# B&R Automation Studio project ARuser
Automation Studio 4.10.4.38 SP; technology packages: mapp 5.17.0, mappView 5.17.0

## Configuration PC

CPU PC_any, AutomationRuntime D4.91, Build 4.1.2, Safety 0.0, Vc V4.52.0

### Task classes (Cpu.sw)
```
Cyclic#1 (cycle 10000 us):
  UserManage <- UserManagement.prg
Binaries: mvLoader, TCData, udbdef, User, asfw, OpcUaMap, iomap, sysconf, arconfig, ashwd, Role, ashwac
Libraries: ArUser, runtime, asieccon, astime, fileio, AsBrStr
```

### Hardware
```
PC : PC_any v1.1.1.0 (OrderNumber=PC)
  Connector IF3:
    InaPort = 11159
  ConfigurationID = ARuser_PC
  VolatileGlobalPvSize = 200000
  Cyclic1Duration = 10000
  Cyclic3Tolerance = 60000000
  Cyclic8Duration = 10000
  FileDevice1
  FileDeviceName1 = FileDevice
  FileDevicePath1 = C:\Users\hendricksf\Desktop
  ActivateOpcUa = 1
  OpcUaInformationModels_PV_Version = 1
```

### Config.mpuserx - PC/mappServices/Config.mpuserx
```
Element UserMgmtX (Type=mpuserx)
  Mgr:
    EditSameLevel = TRUE
  ServerSettings:
    Server:
      AdditionalUserData:
        [0] = mail
        [1] = telephoneNumber
  Users:
    DefUser#1:
      id = Anonymous
      name = 
    DefUser#2:
      id = Bob
      name = Bob Ross
    DefUser#3:
      id = Dave
      name = Dave Chapelle
    DefUser#4:
      id = John
      name = John Doe
  Groups:
    DefGroup#1:
      id = Everyone
      level = 1
    DefGroup#2:
      id = Operator
      level = 2
    DefGroup#3:
      id = Service
      level = 5
    DefGroup#4:
      id = Administrators
      admin = TRUE
```

## Configuration X20CP

CPU X20CP3585, AutomationRuntime D4.91, Build 4.1.2, Vc V4.52.0

### Task classes (Cpu.sw)
```
Cyclic#8:
  UserManage <- mappUser.UserManagement.prg
  RFIDdevice <- mappUser.RFIDdevice.prg
Libraries: runtime, standard, dvframe, sys_lib, AsUSB
```

### Task classes (Cpu.sw)
```
Cyclic#8:
  UserManage <- mappUser.UserManagement.prg
  RFIDdevice <- mappUser.RFIDdevice.prg
Binaries: mvLoader, udbdef, TCData, arconfig, User, Role, Config, iomap, asfw, ashwac, ashwd, sysconf
Libraries: runtime, standard, dvframe, sys_lib, AsUSB, operator, astime, AsIecCon, ArUser, AsBrStr, IecCheck, arssl, fileio, MpUserX, MpBase
```

### Hardware
```
X20CP3585 : X20CP3585 v1.5.0.0
  Connector IF2:
    ActivateDevice = 1
  ConfigurationID = ARuser_X20CP
  UserPartitionSize = 16
  VolatileGlobalPvSize = 120000
  ActivateOpcUa = 1
  OpcUaInformationModels_PV_Version = 1
```

## Logical view

Binary libraries used (declarations not repeated): operator, runtime, astime, AsIecCon, ArUser, AsBrStr, dvframe, AsUSB, sys_lib, standard, IecCheck, MpUserX 5.17.0, MpBase 5.17.0

### Global.typ - Globale Datentypen
```iecst
TYPE
	UserManagementEnum :
		(
		IdleState,
		DestroyListState,
		CreateUserState,
		DeleteUserState,
		ExportListState,
		ImportListState,
		ChangePasswordState,
		ComparePasswordState,
		CreateUserListGetNextState,
		CreateUserListGetFirstState,
		AssignRoleState,
		RoleListMainState,
		RoleListDeleteListState,
		RoleListInitListState,
		ErrorState,
		CreateRoleListGetFirstState,
		CreateRoleListGetNextState,
		RoleListGetNextState
		);
	typUSER : 	STRUCT
		CMD : typUSER_CMD;
		PAR : typUSER_PAR;
		DAT : typUSER_DAT;
		VIS : typUSER_VIS;
		ERR : typUSER_ERR;
	END_STRUCT;
	typUSER_CMD : 	STRUCT
		UserCreate : BOOL;
		UserDelete : BOOL;
		PasswordChange : BOOL;
		RoleCreate : BOOL;
		RoleDelete : BOOL;
		RoleAssign : BOOL;
		Import : BOOL;
		Export : BOOL;
		ListRefresh : BOOL;
		ErrorReset : BOOL;
	END_STRUCT;
	typUSER_PAR : 	STRUCT
		FilePath : STRING[80];
		UserName : STRING[40];
		UserRole : STRING[40];
		Password : STRING[40];
		PasswordRepeat : STRING[40];
		NumberOfUsers : USINT;
	END_STRUCT;
	typUSER_DAT : 	STRUCT
		Users : ARRAY[0..MaxUserNames]OF typUSER_DETAILS;
		Roles : ARRAY[0..MaxUserRoles]OF STRING[40];
		Status : STRING[80];
	END_STRUCT;
	typUSER_VIS : 	STRUCT
		ListUsers : ARRAY[0..MaxUserNames]OF STRING[80];
		ListUserIndex : UINT;
		ListUserRole : ARRAY[0..MaxUserRoles]OF STRING[80];
		ListUserRoleIndex : UINT;
		ListRoles : ARRAY[0..MaxUserRoles]OF STRING[80];
		ListRoleIndex : UINT;
	END_STRUCT;
	typUSER_ERR : 	STRUCT
		Number : DINT;
		State : UserManagementEnum;
	END_STRUCT;
	typUSER_DETAILS : 	STRUCT
		Roles : ARRAY[0..9]OF STRING[40];
		Name : STRING[40];
	END_STRUCT;
END_TYPE
```

### Global.var - Globale Variablen
```iecst
VAR
	ArUser : typUSER; (*Type for user data management*)
END_VAR
VAR CONSTANT
	MaxUserRoles : USINT := 20;
	MaxUserNames : USINT := 50;
END_VAR
```

### Package Logical/Libraries - Globale Bibliotheken

- Visualisation Logical/mappView (not shown)

### UserTypes.typ
```iecst
TYPE
	ClientInfoType : 	STRUCT
		userId : WSTRING[80];
		isValid : BOOL;
		ipAddress : WSTRING[15];
		languageId : WSTRING[2];
		screenResolution : WSTRING[32];
		slotId : SINT;
	END_STRUCT;
	rfidManagementEnum :
		(
		IdleRFID, (*Search for reader or new tokens*)
		SetToken, (*Assign token to user*)
		SetPassword, (*Set token as user password*)
		DeleteToken, (*Delete token from user*)
		IdentifyToken, (*Identify token*)
		CreateNodeList, (* Create a list of Node-IDs from all active USB devices*)
		ReadDeviceData, (* Read out the specific data from the Node-IDs*)
		CheckDevice, (* Check RFID reader data*)
		OpenDevice, (*Open serial communication*)
		InitDevice, (*Send inital data to setup RFID reader*)
		DataWrite, (*Send data to RFID reader*)
		DataRead, (*Read data from RFID reader*)
		CloseDevice, (*Close serial connection*)
		ErrorRFID (*Error state*)
		);
	enumRFIDtype :
		(
		RFID_5E9010_29,
		RFID_5E9030_29,
		RFID_NONE
		);
	rfidCMD : 	STRUCT
		ReaderEnable : BOOL; (*Scan USB ports automatically*)
		TokenAssign : BOOL;
		TokenRemove : BOOL;
		ErrorReset : BOOL; (*Reset error*)
	END_STRUCT;
	rfidPAR : 	STRUCT
		RefreshInterval : UINT; (*Intervall timer for USB device refresh*)
		DataMinLen : UDINT;
		AutoLogin : BOOL;
		UserName : STRING[40];
		Password : STRING[40];
	END_STRUCT;
	rfidDAT : 	STRUCT
		IsConnected : BOOL; (*Shows if a USB stick is connected*)
		Type : enumRFIDtype := RFID_NONE;
		Data : STRING[80];
		Cnt : UDINT;
		Status : STRING[80];
	END_STRUCT;
	rfidVIS : 	STRUCT
		ExecuteLogin : BOOL;
		ShowMessageBoxOK : BOOL;
	END_STRUCT;
	rfidERR : 	STRUCT
		Number : DINT;
		State : rfidManagementEnum;
	END_STRUCT;
	rfidMAIN : 	STRUCT
		CMD : rfidCMD; (*Command structure*)
		PAR : rfidPAR; (*Parameter structure*)
		DAT : rfidDAT;
		VIS : rfidVIS; (*Error structure*)
		ERR : rfidERR; (*Error structure*)
	END_STRUCT;
	userManagementEnum :
		(
		IdleUser, (*Wait state*)
		DestroyList,
		CreateUser,
		DeleteUser,
		RenameUser,
		ExportList,
		ImportList,
		ChangePassword,
		ComparePassword,
		CreateUserListGetNext,
		CreateUserListGetFirst,
		AssignRole,
		ReleaseRole,
		RoleListMain,
		RoleListDeleteList,
		RoleListInitList,
		CreateRoleListGetFirst,
		CreateRoleListGetNext,
		RoleListGetNext,
		PropertyRead,
		PropertyWrite,
		ErrorUser
		);
	userMAIN : 	STRUCT
		CMD : userCMD;
		PAR : userPAR;
		DAT : userDAT;
		VIS : ARRAY[0..MAX_USER_CLIENTS]OF userVIS;
		ERR : userERR;
	END_STRUCT;
	userCMD : 	STRUCT
		UserCreate : BOOL;
		UserDelete : BOOL;
		UserRename : BOOL;
		PasswordChange : BOOL;
		RoleAssign : BOOL;
		RoleRemove : BOOL;
		Import : BOOL;
		Export : BOOL;
		ListRefresh : BOOL;
		ErrorReset : BOOL;
	END_STRUCT;
	userPAR : 	STRUCT
		FilePath : STRING[100] := 'F:/UserDataExport.txt';
		UserName : STRING[MAX_USER_ITEM_LEN];
		UserNameNew : STRING[MAX_USER_ITEM_LEN];
		UserRole : STRING[MAX_USER_ITEM_LEN];
		Password : STRING[MAX_USER_ITEM_LEN];
		PasswordRepeat : STRING[MAX_USER_ITEM_LEN];
		VisuSlotID : USINT;
	END_STRUCT;
	userDAT : 	STRUCT
		Users : ARRAY[0..MAX_USER_NAMES]OF userDETAILS;
		Roles : ARRAY[0..MAX_USER_ROLES]OF STRING[MAX_USER_ITEM_LEN];
		Status : STRING[200];
		UserActive : ARRAY[0..MAX_USER_CLIENTS]OF STRING[MAX_USER_ITEM_LEN];
	END_STRUCT;
	userVIS : 	STRUCT
		ListUsers : ARRAY[0..MAX_USER_NAMES]OF STRING[MAX_USER_ITEM_LEN];
		ListUserIndex : UINT;
		ListUserValue : STRING[MAX_USER_ITEM_LEN];
		ListUserRole : ARRAY[0..MAX_USER_ROLES]OF STRING[MAX_USER_ITEM_LEN];
		ListUserRoleIndex : UINT;
		ListRoles : ARRAY[0..MAX_USER_ROLES]OF STRING[MAX_USER_ITEM_LEN];
		ListRoleIndex : UINT;
		RoleDeleteEnabled : BOOL;
		UserDeleteEnabled : BOOL;
		ShowMessageBoxOK : BOOL;
		ShowMessageBoxError : BOOL;
	END_STRUCT;
	userERR : 	STRUCT
		No : DINT;
		State : userManagementEnum;
		Text : STRING[100];
	END_STRUCT;
	userDETAILS : 	STRUCT
		Roles : ARRAY[0..MAX_USER_ROLES]OF STRING[MAX_USER_ITEM_LEN];
		Name : STRING[MAX_USER_ITEM_LEN];
	END_STRUCT;
END_TYPE
```

### UserVariables.var
```iecst
(*Global constants*)
VAR CONSTANT
	RFID_TYPE : enumRFIDtype := RFID_5E9030_29;
END_VAR
(*Global variable structure*)
VAR
	ArUser : userMAIN; (*Type for user data management*)
	RFID : rfidMAIN;
END_VAR
```

### Program Logical/mappUser/UserManagement (IEC)

#### Main.st - Init, cyclic, exit code
```iecst
// --------------------------------------------------------------------------------------------------------------------
// General user task. This is a support task for the mappView visualization. The following functions are implemneted
// - Export and import user data
// Version 2.0
// --------------------------------------------------------------------------------------------------------------------
PROGRAM _INIT
END_PROGRAM

PROGRAM _CYCLIC

	FOR override:=0 TO MAX_CYCLES DO
		// --------------------------------------------------------------------------------------------------------------------
		// User managment state machine
		// --------------------------------------------------------------------------------------------------------------------
		CASE UserManagementState OF
			// --------------------------------------------------------------------------------------------------------------------
			// Wait for new command
			// --------------------------------------------------------------------------------------------------------------------
			IdleUser:

				// --------------------------------------------------------------------------------------------------------------------
				// Rename user
				IF (ArUser.CMD.Export) THEN
					ArUserExport_0(Execute := FALSE);
					UserManagementState := ExportList;
					// Import user data
				ELSIF (ArUser.CMD.Import) THEN
					ArUserImport_0(Execute := FALSE);
					UserManagementState := ImportList;
				END_IF;

				// --------------------------------------------------------------------------------------------------------------------
				// Reset fields on new command
				ArUser.CMD.ErrorReset := FALSE;

				// --------------------------------------------------------------------------------------------------------------------
				// Export user list to file
				// --------------------------------------------------------------------------------------------------------------------
			ExportList:
				ArUserExport_0(Execute := TRUE, FilePath := ArUser.PAR.FilePath);

				// --------------------------------------------------------------------------------------------------------------------
				// Success
				IF ArUserExport_0.Done AND NOT ArUserExport_0.Busy THEN
					ArUser.Status := 'Export finished';
					ArUser.CMD.Export := FALSE;
					UserManagementState := IdleUser;
					// Error
				ELSIF ArUserExport_0.Error THEN
					ArUser.ERR.No := ArUserExport_0.ErrorID;
					ArUser.ERR.State := UserManagementState;
					UserManagementState := ErrorUser;
				END_IF;

				// --------------------------------------------------------------------------------------------------------------------
				// Import user list from file
				// --------------------------------------------------------------------------------------------------------------------
			ImportList:
				ArUserImport_0(Execute := TRUE, FilePath := ArUser.PAR.FilePath);

				// --------------------------------------------------------------------------------------------------------------------
				// Success
				IF ArUserImport_0.Done AND NOT ArUserImport_0.Busy THEN
					ArUser.Status := 'Import finished';
					ArUser.CMD.Import := FALSE;
					UserManagementState := IdleUser;
					// Error
				ELSIF ArUserImport_0.Error THEN
					ArUser.ERR.No := ArUserImport_0.ErrorID;
					ArUser.ERR.State := UserManagementState;
					UserManagementState := ErrorUser;
				END_IF;

				// --------------------------------------------------------------------------------------------------------------------
				// Error
				// --------------------------------------------------------------------------------------------------------------------
			ErrorUser:
				// --------------------------------------------------------------------------------------------------------------------
				// Reset function blocks
				ArUserImport_0(Execute := FALSE);
				ArUserExport_0(Execute := FALSE);

				// --------------------------------------------------------------------------------------------------------------------
				// Generate text for most common errors
				IF(ArUser.ERR.No = arUSER_ERR_PARAMETER) THEN
					ArUser.Status := 'ERR: path is empty';
				ELSE
					ArUser.Status := 'Error executing command';
				END_IF
				// --------------------------------------------------------------------------------------------------------------------
				// Return to idle state
				IF ArUser.CMD.ErrorReset THEN

					brsmemset(ADR(ArUser.ERR), 0, SIZEOF(ArUser.ERR));
					ArUser.CMD.ErrorReset := FALSE;
					UserManagementState := IdleUser;
				END_IF;
				brsmemset(ADR(ArUser.CMD), 0, SIZEOF(ArUser.CMD));
				RETURN;
		END_CASE;
	END_FOR;

END_PROGRAM
```

#### Variables.var - Local variables
```iecst
(*General*)
VAR
	UserManagementState : userManagementEnum := IdleUser; (*State Machine for UserManagementState*)
	ArUserExport_0 : ArUserExport; (*Export all user and role data*)
	ArUserImport_0 : ArUserImport; (*Import all user and role data*)
	override : USINT;
END_VAR
VAR CONSTANT
	MAX_CYCLES : USINT := 10; (*Maximum number of override cycles*)
END_VAR
```

#### LocalFunctions.fun
```iecst
{REDUND_ERROR} FUNCTION String2DataProvider : BOOL (*create mappView string data provider*) (*$GROUP=User,$CAT=User,$GROUPICON=User.png,$CATICON=User.png*)
	VAR_INPUT
		SourceString : UDINT;
		TargetString : UDINT;
	END_VAR
END_FUNCTION
```

### Program Logical/mappUser/RFIDdevice (IEC) - Sample for all AsUSB-Library-Functions

#### RFIDdevice.st - Cyclic code
```iecst
// --------------------------------------------------------------------------------------------------------------------
// This task allows user login with RFID tokens. The following functions are implemneted
// - Assign or remove token from user
// Version 1.1
// -----------------------------------------------------------------------------------------------------------
PROGRAM _INIT
	// -----------------------------------------------------------------------------------------------------------
	// Start auto scan, set default parameters
	RFID.CMD.ReaderEnable := TRUE;				// AutoScan for RFID reader and token data
	RFID.PAR.AutoLogin := TRUE;					// Auto login user when token is detected
	RFID.PAR.RefreshInterval := 50;				// Read data every 500ms
	RFID.PAR.DataMinLen := 16;					// Mimimum length of RFID data, everything shorter will be ignored

	// -----------------------------------------------------------------------------------------------------------
	// Use mappUser sample variables when it exists
	PV_xgetadr(ADR('ArUser.PAR.UserName'), ADR(ArUserNameAdr), ADR(ArUserNameLen));
	PV_xgetadr(ADR('ArUser.PAR.Password'), ADR(ArUserPasswordAdr), ADR(ArUserPasswordLen));

END_PROGRAM

PROGRAM _CYCLIC

	CASE rfid_state OF
		// -----------------------------------------------------------------------------------------------------------
		// IdleRFID state
		// -----------------------------------------------------------------------------------------------------------
		IdleRFID:
			// --------------------------------------------------------------------------------------------------------------------
			// Remove token from user
			IF RFID.CMD.TokenRemove THEN
				ArUserSetToken_0(Execute := FALSE);
				RFID.PAR.Password := RFID.PAR.UserName;
				rfid_state := SetToken;
			END_IF

			// Refresh USB data when enabled
			IF RFID.CMD.ReaderEnable THEN
				// --------------------------------------------------------------------------------------------------------------------
				// Get new RFID data
				TimerAutoScan(IN:=1, PT:=RFID.PAR.RefreshInterval);
				IF TimerAutoScan.Q THEN
					TimerAutoScan(IN:=0);
					node := 0;
					IF(RFID.DAT.IsConnected) THEN
						// Reader 5E9010.29 needs a request before reading token data
						IF(RFID.DAT.Type = RFID_5E9010_29) THEN
							data_write := REQ_ACTIVE;
							callback := IdleRFID;
							rfid_state := DataWrite;
						// Make sure reader 5E9030 is still connected
						ELSE
							brsmemset(ADR(usb_data), 0, SIZEOF(usb_data));
							rfid_state := CreateNodeList;
						END_IF
					// Search for RFID reader when not connected
					ELSE
						brsmemset(ADR(usb_data), 0, SIZEOF(usb_data));
						rfid_state := CreateNodeList;
					END_IF
				END_IF

				// --------------------------------------------------------------------------------------------------------------------
				// When RFID reader is connected
				IF RFID.DAT.IsConnected = TRUE THEN
					// --------------------------------------------------------------------------------------------------------------------
					// Assign token to user
					IF RFID.CMD.TokenAssign THEN
						RFID.PAR.Password := RFID.DAT.Data;
						ArUserSetToken_0(Execute := FALSE);
						rfid_state := SetToken;
					END_IF

					// --------------------------------------------------------------------------------------------------------------------
					// Read data from serial device
					FRM_read_0.ident := FRM_xopen_0.ident;
					FRM_read_0.enable := 1;
					FRM_read_0();
					TimerTimeout(IN:=1, PT:=2*RFID.PAR.RefreshInterval);

					// --------------------------------------------------------------------------------------------------------------------
					// New data arrived
					IF FRM_read_0.status = 0 THEN
						// Reset timer and buffer
						TimerTimeout(IN:=0);
						brsmemset(ADR(data_read), 0, SIZEOF(data_read));
						brsmemcpy(ADR(data_read), FRM_read_0.buffer, FRM_read_0.buflng);

						// Make sure data is valid
						IF RFID.DAT.IsConnected AND brsmemcmp(ADR(data_read), ADR('[,'), 2) <> 0 AND brsmemcmp(ADR(data_read), ADR('PiccRemove:'), 11) <> 0 THEN
							// Remove unwanted characters from token data
							idx := 0;
							REPEAT
								IF(brsmemcmp(ADR(data_read), ADR('PiccSelect:'), 11) = 0) THEN
									brsmemcpy(ADR(data_read)+idx, ADR(data_read)+idx+11, brsstrlen(ADR(data_read))-idx);
								ELSIF(brsmemcmp(ADR(data_read)+idx, ADR(' '), 1) = 0) THEN
									brsmemcpy(ADR(data_read)+idx, ADR(data_read)+idx+1, brsstrlen(ADR(data_read))-idx);
								ELSIF(brsmemcmp(ADR(data_read)+idx, ADR('['), 1) = 0) THEN
									brsmemcpy(ADR(data_read)+idx, ADR(data_read)+idx+1, brsstrlen(ADR(data_read))-idx);
								ELSIF(brsmemcmp(ADR(data_read)+idx, ADR(']'), 1) = 0) THEN
									brsmemcpy(ADR(data_read)+idx, ADR(data_read)+idx+1, brsstrlen(ADR(data_read))-idx);
								ELSIF(brsmemcmp(ADR(data_read)+idx, ADR('$r'), 1) = 0) THEN
									brsmemcpy(ADR(data_read)+idx, ADR(data_read)+idx+1, brsstrlen(ADR(data_read))-idx);
								ELSIF(brsmemcmp(ADR(data_read)+idx, ADR('$n'), 1) = 0) THEN
									brsmemcpy(ADR(data_read)+idx, ADR(data_read)+idx+1, brsstrlen(ADR(data_read))-idx);
								ELSIF(brsmemcmp(ADR(data_read)+idx, ADR(','), 1) = 0) THEN
									brsmemset(ADR(data_read)+idx, 0, brsstrlen(ADR(data_read))-idx);
								ELSE
									idx := idx + 1;
								END_IF
								UNTIL idx = FRM_read_0.buflng
							END_REPEAT;

							// Check RFID data size
							IF brsstrlen(ADR(data_read)) >= RFID.PAR.DataMinLen THEN
								// Maintain stats, move data, identify token
								RFID.DAT.Cnt := RFID.DAT.Cnt + 1;
								RFID.VIS.ExecuteLogin := FALSE;
								brsmemset(ADR(RFID.DAT.Data), 0, SIZEOF(RFID.DAT.Data));
								brsstrcpy(ADR(RFID.DAT.Data), ADR(data_read));
								ArUserAuthToken_0(Execute := FALSE);
								IF(brsstrcmp(ADR(tmpTokenOld), ADR(RFID.DAT.Data)) <> 0) THEN
									rfid_state := IdentifyToken;
								END_IF
								tmpTokenOld := RFID.DAT.Data;
							END_IF
						// Reset old token when it was removed from reader
						ELSIF RFID.DAT.IsConnected AND brsmemcmp(ADR(data_read), ADR('PiccRemove:'), 11) = 0 THEN
							tmpTokenOld := '';
						END_IF

						// Release read buffer
						FRM_rbuf_0.buffer := FRM_read_0.buffer;
						FRM_rbuf_0.buflng := FRM_read_0.buflng;
						FRM_rbuf_0.ident := FRM_xopen_0.ident;
						FRM_rbuf_0.enable := 1;
						FRM_rbuf_0();
					// Read response timeout
					ELSIF TimerTimeout.Q THEN
						// Ignore timeout for 5E9030
						IF RFID.DAT.Type <> RFID_5E9030_29 THEN
							RFID.ERR.Number := 50020;
							RFID.DAT.Status := 'Read response timeout';
							rfid_state := ErrorRFID;
						END_IF
					// Cyclic read error
					ELSIF FRM_read_0.status <> frmERR_NOINPUT AND FRM_read_0.status <> ERR_FUB_BUSY THEN
						RFID.ERR.Number := FRM_read_0.status;
						RFID.DAT.Status := 'Error in cyclic read';
						rfid_state := ErrorRFID;
					END_IF
				ELSE
					RFID.CMD.TokenAssign := FALSE;
				END_IF

			// --------------------------------------------------------------------------------------------------------------------
			// Close USB connection
			ELSIF RFID.DAT.IsConnected = TRUE THEN
				rfid_state := CloseDevice;

			// --------------------------------------------------------------------------------------------------------------------
			// Function is disabled
			ELSE
				RFID.CMD.TokenAssign := FALSE;
				TimerAutoScan(IN:=0);
				RFID.DAT.Status := 'Disabled';
			END_IF;

			// --------------------------------------------------------------------------------------------------------------------
			// Reset old data
			IF RFID.DAT.Data = '' THEN
				tmpTokenOld := RFID.DAT.Data;
			END_IF

			// --------------------------------------------------------------------------------------------------------------------
			// Reset error
			IF RFID.CMD.ErrorReset  THEN
				brsmemset(ADR(RFID.DAT.Data), 0, SIZEOF(RFID.DAT.Data));
				RFID.CMD.ErrorReset := FALSE;
			END_IF
		// --------------------------------------------------------------------------------------------------------------------
		// Set user token
		// --------------------------------------------------------------------------------------------------------------------
		SetToken:
			ArUserSetToken_0(Execute := TRUE , UserName := RFID.PAR.UserName, Token := RFID.PAR.Password);

			// --------------------------------------------------------------------------------------------------------------------
			// Success
			IF ArUserSetToken_0.Done AND NOT ArUserSetToken_0.Busy THEN
				ArUserSetPassword_0(Execute := FALSE);
				rfid_state := SetPassword;
			// Error
			ELSIF ArUserSetToken_0.Error THEN
				RFID.DAT.Status := 'Error assigning token';
				RFID.ERR.Number := ArUserSetToken_0.ErrorID;
				RFID.ERR.State := rfid_state;
				rfid_state := ErrorRFID;
			END_IF;

		// --------------------------------------------------------------------------------------------------------------------
		// Set password to token data
		// --------------------------------------------------------------------------------------------------------------------
		SetPassword:
			ArUserSetPassword_0(Execute := TRUE , UserName := RFID.PAR.UserName , Password := RFID.PAR.Password);

			// --------------------------------------------------------------------------------------------------------------------
			// Success
			IF ArUserSetPassword_0.Done AND NOT ArUserSetPassword_0.Busy THEN
				IF(RFID.CMD.TokenAssign) THEN
					RFID.DAT.Status := 'Token was assigned to user ';
					brsstrcat(ADR(RFID.DAT.Status), ADR(RFID.PAR.UserName));
					RFID.CMD.TokenAssign := FALSE;
				ELSE
					RFID.DAT.Status := 'Token was removed from user ';
					brsstrcat(ADR(RFID.DAT.Status), ADR(RFID.PAR.UserName));
					brsstrcat(ADR(RFID.DAT.Status), ADR(' password is set to '));
					brsstrcat(ADR(RFID.DAT.Status), ADR(RFID.PAR.Password));
					RFID.CMD.TokenRemove := FALSE;
				END_IF
				RFID.VIS.ShowMessageBoxOK := TRUE;
				rfid_state := IdleRFID;
			// Error
			ELSIF ArUserSetPassword_0.Error THEN
				RFID.DAT.Status := 'Error setting user password';
				RFID.ERR.Number := ArUserSetPassword_0.ErrorID;
				RFID.ERR.State := rfid_state;
				rfid_state := ErrorRFID;
			END_IF;

		// --------------------------------------------------------------------------------------------------------------------
		// Identify user token
		// --------------------------------------------------------------------------------------------------------------------
		IdentifyToken:
			ArUserAuthToken_0(Execute := TRUE, Token := RFID.DAT.Data);

			// --------------------------------------------------------------------------------------------------------------------
			// Success
			IF ArUserAuthToken_0.Done AND NOT ArUserAuthToken_0.Busy THEN
				IF ArUserAuthToken_0.IsAuthentic THEN
					RFID.PAR.UserName := ArUserAuthToken_0.UserName;
					RFID.PAR.Password := ArUserAuthToken_0.Token;
					RFID.DAT.Status := 'Token from user ';
					brsstrcat(ADR(RFID.DAT.Status), ADR(RFID.PAR.UserName));
					brsstrcat(ADR(RFID.DAT.Status), ADR(' identified'));
					// Transfer user name and password from ArUser template when it exists
					IF(ArUserNameAdr <> 0 AND ArUserPasswordAdr <> 0) THEN
						brsstrcpy(ArUserNameAdr, ADR(RFID.PAR.UserName));
						brsstrcpy(ArUserPasswordAdr, ADR(RFID.PAR.Password));
					END_IF
					IF(RFID.PAR.AutoLogin) THEN
						RFID.VIS.ExecuteLogin := TRUE;
						brsstrcat(ADR(RFID.DAT.Status), ADR(' and logged in'));
					END_IF
				ELSE
					RFID.DAT.Status := 'Token is not assigned to any user ';
					RFID.VIS.ShowMessageBoxOK := TRUE;
				END_IF
				rfid_state := IdleRFID;
				// Error
			ELSIF ArUserAuthToken_0.Error THEN
				RFID.DAT.Status := 'Error identifying token';
				RFID.ERR.Number := ArUserAuthToken_0.ErrorID;
				RFID.ERR.State := rfid_state;
				rfid_state := ErrorRFID;
			END_IF;

		// -----------------------------------------------------------------------------------------------------------
		// Get USB device list
		// -----------------------------------------------------------------------------------------------------------
		CreateNodeList:
			UsbNodeListGet_0.enable := 1;
			UsbNodeListGet_0.pBuffer := ADR(node_id_buffer);
			UsbNodeListGet_0.bufferSize := SIZEOF(node_id_buffer);
			UsbNodeListGet_0.filterInterfaceClass := 0;
			UsbNodeListGet_0.filterInterfaceSubClass := 0;
			UsbNodeListGet_0;

			// --------------------------------------------------------------------------------------------------------------------
			// Success
			IF UsbNodeListGet_0.status = 0 THEN
				rfid_state := ReadDeviceData;
			// No USB devices found
			ELSIF UsbNodeListGet_0.status = asusbERR_USB_NOTFOUND THEN
				// Unlink old device if it is gone now otherwise report error
				IF(RFID.DAT.IsConnected) THEN
					rfid_state := CloseDevice;
				ELSE
					RFID.ERR.Number := UsbNodeListGet_0.status;
					RFID.DAT.Status := 'No USB reader detected';
					rfid_state := ErrorRFID;
				END_IF
			// Error
			ELSIF UsbNodeListGet_0.status <> ERR_FUB_BUSY THEN
				RFID.DAT.Status := 'Error generating USB node list';
				RFID.ERR.Number := UsbNodeListGet_0.status;
				RFID.ERR.State := rfid_state;
				rfid_state := ErrorRFID;
			END_IF;

		// -----------------------------------------------------------------------------------------------------------
		// Get device information
		// -----------------------------------------------------------------------------------------------------------
		ReadDeviceData:
			UsbNodeGet_0.enable := 1;
			UsbNodeGet_0.nodeId := node_id_buffer[node];
			UsbNodeGet_0.pBuffer := ADR(usb_data[node]);
			UsbNodeGet_0.bufferSize := SIZEOF (usb_data[node]);
			UsbNodeGet_0;

			// --------------------------------------------------------------------------------------------------------------------
			// Success
			IF UsbNodeGet_0.status = 0 THEN
				// Make sure we have enough space to store USB data, proceed with next rfid_state when all devices are detetced
				IF (node = UsbNodeListGet_0.listNodes - 1) OR (node > SIZEOF(usb_data)/SIZEOF(usb_data[0])) THEN
					idx := 0;
					rfid_state := CheckDevice;
				// Get next USB device
				ELSE
					node := node + 1;
				END_IF;
			// Error
			ELSIF UsbNodeGet_0.status <> ERR_FUB_BUSY THEN
				RFID.ERR.Number := UsbNodeGet_0.status;
				RFID.ERR.State := rfid_state;
				rfid_state := ErrorRFID;
			END_IF;

		// -----------------------------------------------------------------------------------------------------------
		// Check if device is connected
		// -----------------------------------------------------------------------------------------------------------
		CheckDevice:
			// Check if device is already linked
			IF RFID.DAT.IsConnected THEN
				// Device is already linked, return to IdleRFID state
				IF brsmemcmp(ADR(usb_data_linked), ADR(usb_data[idx]), SIZEOF(usb_data[idx])) = 0 THEN
					rfid_state := IdleRFID;
				// Check next device
				ELSIF idx < node THEN
					idx := idx + 1;
				// Reader was disconnected
				ELSE
					RFID.DAT.Status := 'Reader disconnected';
					RFID.DAT.IsConnected := FALSE;
					RFID.ERR.Number := ERR_RFID_DISCONNECTED;
					RFID.ERR.State := rfid_state;
					rfid_state := ErrorRFID;
				END_IF
			ELSE
				// Device is RFID reader type 5E9010.29
				IF usb_data[idx].productId = DEV_PRODUCT_ID[RFID_5E9010_29] AND usb_data[idx].vendorId = DEV_VENDOR_ID[RFID_5E9010_29] THEN
					// Copy configuration data and request string
					brsmemcpy(ADR(usb_data_linked), ADR(usb_data[idx]), SIZEOF(usb_data_linked));
					brsmemset(ADR(CFG_ACTIVE), 0, SIZEOF(CFG_ACTIVE));
					brsmemcpy(ADR(CFG_ACTIVE), ADR(CFG_5E9010_29), SIZEOF(CFG_5E9010_29));
					REQ_ACTIVE := REQ_5E9010_29;
					RFID.DAT.Type := RFID_5E9010_29;
					RFID.DAT.Status := 'Reader 5E9010 connected';
					rfid_state := OpenDevice;
					// Device is RFID reader type 5E9030.29
				ELSIF usb_data[idx].productId = DEV_PRODUCT_ID[RFID_5E9030_29] AND usb_data[idx].vendorId = DEV_VENDOR_ID[RFID_5E9030_29] THEN
					// Copy configuration data and request string
					brsmemcpy(ADR(usb_data_linked), ADR(usb_data[idx]), SIZEOF(usb_data_linked));
					brsmemset(ADR(CFG_ACTIVE), 0, SIZEOF(CFG_ACTIVE));
					brsmemcpy(ADR(CFG_ACTIVE), ADR(CFG_5E9030_29), SIZEOF(CFG_5E9030_29));
					RFID.DAT.Type := RFID_5E9030_29;
					RFID.DAT.Status := 'Reader 5E9030 connected';
					rfid_state := OpenDevice;
				ELSE
					IF idx < node THEN
						idx := idx + 1;
					ELSE
						RFID.DAT.Status := 'No USB reader detected';
						rfid_state := IdleRFID;
					END_IF
				END_IF
			END_IF

		// -----------------------------------------------------------------------------------------------------------
		// Open device
		// -----------------------------------------------------------------------------------------------------------
		OpenDevice:
			// Open serial device communication
			FRM_xopen_0.device := ADR(usb_data_linked.ifName);
			FRM_xopen_0.enable := 1;
			FRM_xopen_0();

			// --------------------------------------------------------------------------------------------------------------------
			// Success
			IF FRM_xopen_0.status = 0 THEN
				rfid_init := 0;
				rfid_state := InitDevice;
			// Error
			ELSIF FRM_xopen_0.status <> ERR_FUB_BUSY THEN
				rfid_state := ErrorRFID;
			END_IF;

		// -----------------------------------------------------------------------------------------------------------
		// Init RFID
		// -----------------------------------------------------------------------------------------------------------
		InitDevice:
			// Send next configuration data
			IF CFG_ACTIVE[rfid_init] <> '' THEN
				data_write := CFG_ACTIVE[rfid_init];
				callback := InitDevice;
				rfid_init := rfid_init + 1;
				rfid_state := DataWrite;
			// Finish sending configuration
			ELSE
				RFID.DAT.IsConnected := TRUE;
				rfid_state := IdleRFID;
			END_IF;

		// -----------------------------------------------------------------------------------------------------------
		// Empty read buffer before sending next command
		// -----------------------------------------------------------------------------------------------------------
		DataWrite:
			// Write data to serial device
			FRM_write_0.buffer := ADR(data_write);
			FRM_write_0.buflng := UDINT_TO_UINT(brsstrlen(ADR(data_write)));
			FRM_write_0.ident := FRM_xopen_0.ident;
			FRM_write_0.enable := 1;
			FRM_write_0();

			// --------------------------------------------------------------------------------------------------------------------
			// Success
			IF FRM_write_0.status = 0 THEN
				IF RFID.DAT.IsConnected THEN
					rfid_state := callback;
				ELSE
					TimerTimeout(IN:=0);
					rfid_state := DataRead;
				END_IF
			// Error
			ELSIF FRM_write_0.status <> ERR_FUB_BUSY THEN
				FRM_robuf_0.buffer := FRM_write_0.buffer;
				FRM_robuf_0.buflng := FRM_write_0.buflng;
				FRM_robuf_0.ident := FRM_xopen_0.ident;
				FRM_robuf_0.enable := 1;
				rfid_state := ErrorRFID;
			END_IF;

		// -----------------------------------------------------------------------------------------------------------
		// Read data from RFID
		// -----------------------------------------------------------------------------------------------------------
		DataRead:
			// Read data from serial device
			FRM_read_0.ident := FRM_xopen_0.ident;
			FRM_read_0.enable := 1;
			FRM_read_0();
			TimerTimeout(IN:=1, PT:=100);

			// --------------------------------------------------------------------------------------------------------------------
			// Success
			IF FRM_read_0.status = 0 THEN
				TimerTimeout(IN:=0);
				// Make sure data fits into buffer
				IF FRM_read_0.buflng < SIZEOF(data_read) THEN
					brsmemset(ADR(data_write), 0, SIZEOF(data_write));
					brsmemset(ADR(data_read), 0, SIZEOF(data_read));
					brsmemcpy(ADR(data_read), FRM_read_0.buffer, FRM_read_0.buflng);
					// Remove unwanted characters from token data
					idx := 0;
					REPEAT
						IF(brsmemcmp(ADR(data_read)+idx, ADR('['), 1) = 0) THEN
							brsmemcpy(ADR(data_read)+idx, ADR(data_read)+idx+1, brsstrlen(ADR(data_read))-idx);
						ELSIF(brsmemcmp(ADR(data_read)+idx, ADR(' '), 1) = 0) THEN
							brsmemcpy(ADR(data_read)+idx, ADR(data_read)+idx+1, brsstrlen(ADR(data_read))-idx);
						ELSIF(brsmemcmp(ADR(data_read)+idx, ADR('*'), 1) = 0) THEN
							brsmemcpy(ADR(data_read)+idx, ADR(data_read)+idx+1, brsstrlen(ADR(data_read))-idx);
						ELSIF(brsmemcmp(ADR(data_read)+idx, ADR(']'), 1) = 0) THEN
							brsmemcpy(ADR(data_read)+idx, ADR(data_read)+idx+1, brsstrlen(ADR(data_read))-idx);
						ELSIF(brsmemcmp(ADR(data_read)+idx, ADR('$r'), 1) = 0) THEN
							brsmemcpy(ADR(data_read)+idx, ADR(data_read)+idx+1, brsstrlen(ADR(data_read))-idx);
						ELSIF(brsmemcmp(ADR(data_read)+idx, ADR('$n'), 1) = 0) THEN
							brsmemcpy(ADR(data_read)+idx, ADR(data_read)+idx+1, brsstrlen(ADR(data_read))-idx);
						ELSIF(brsmemcmp(ADR(data_read)+idx, ADR(','), 1) = 0) THEN
							brsmemset(ADR(data_read)+idx, 0, brsstrlen(ADR(data_read))-idx);
						ELSE
							idx := idx + 1;
						END_IF
						UNTIL idx = FRM_read_0.buflng
					END_REPEAT;

					// Response for 5E9010 should be empty, Initial response for 5E9030 can be ignored
					IF brsstrcmp(ADR(data_read), ADR('')) = 0 OR RFID.DAT.Type = RFID_5E9030_29 THEN
						rfid_state := callback;
					ELSE
						RFID.ERR.Number := ERR_RFID_RESPONSE;
						RFID.DAT.Status := 'RFID response incorrect';
						rfid_state := ErrorRFID;
					END_IF
				// Read data exceeds buffer
				ELSE
					RFID.ERR.Number := ERR_RFID_BUFFER;
					RFID.DAT.Status := 'Receive buffer exceeds maximum';
					rfid_state := ErrorRFID;
				END_IF
				// Release read buffer
				FRM_rbuf_0.buffer := FRM_read_0.buffer;
				FRM_rbuf_0.buflng := FRM_read_0.buflng;
				FRM_rbuf_0.ident := FRM_xopen_0.ident;
				FRM_rbuf_0.enable := 1;
				FRM_rbuf_0();
			// Error from serial read
			ELSIF FRM_read_0.status <> ERR_FUB_BUSY  AND FRM_read_0.status <> frmERR_NOINPUT THEN
				rfid_state := ErrorRFID;
			// Read response timeout
			ELSIF(TimerTimeout.Q) THEN
				// Ignore timeout for 5E9030
				IF RFID.DAT.Type = RFID_5E9030_29 THEN
					rfid_state := callback;
				ELSE
					RFID.ERR.Number := ERR_RFID_READ_TIMEOUT;
					RFID.DAT.Status := 'Read response timeout';
					rfid_state := ErrorRFID;
				END_IF;
			END_IF;

		// -----------------------------------------------------------------------------------------------------------
		// Close device
		// -----------------------------------------------------------------------------------------------------------
		CloseDevice:
			// Close serial device communication
			FRM_close_0.ident := FRM_xopen_0.ident;
			FRM_close_0.enable := 1;
			FRM_close_0();

			// --------------------------------------------------------------------------------------------------------------------
			// Success
			IF FRM_close_0.status = 0 THEN
				RFID.DAT.IsConnected := FALSE;
				RFID.DAT.Type := RFID_NONE;
				IF(RFID.CMD.ReaderEnable) THEN
					rfid_init := 0;
					rfid_state := InitDevice;
				ELSE
					rfid_state := IdleRFID;
				END_IF
			// Error
			ELSIF FRM_close_0.status <> ERR_FUB_BUSY THEN
				rfid_state := ErrorRFID;
			END_IF;

		// -----------------------------------------------------------------------------------------------------------
		// Error state
		// -----------------------------------------------------------------------------------------------------------
		ErrorRFID:
			// Reset commands
			RFID.CMD.ReaderEnable := FALSE;
			RFID.CMD.TokenAssign := FALSE;
			RFID.CMD.TokenRemove := FALSE;
			RFID.DAT.IsConnected := FALSE;

			// Reset error
			IF RFID.CMD.ErrorReset THEN
				FRM_close_0.ident := FRM_xopen_0.ident;
				FRM_close_0.enable := 1;
				FRM_close_0();

				brsmemset(ADR(RFID.ERR), 0, SIZEOF(RFID.ERR));
				brsmemset(ADR(RFID.DAT), 0, SIZEOF(RFID.DAT));
				RFID.CMD.ErrorReset := FALSE;
				rfid_state := IdleRFID;
			END_IF
	END_CASE;

END_PROGRAM

PROGRAM _EXIT
	REPEAT
		FRM_close_0.ident := FRM_xopen_0.ident;
		FRM_close_0.enable := 1;
		FRM_close_0();

		UNTIL FRM_close_0.status <> ERR_FUB_BUSY
	END_REPEAT;
END_PROGRAM
```

#### RFIDdevice.var - Data for read_data Task
```iecst
(*----------------------------------------------------------------------------------------------------------------------------------------------------------------------------------------------------------------------------------------------------------------------*)
(*Local functions*)
VAR
	TimerAutoScan : TON_10ms; (*Scan timer for tokens*)
	TimerTimeout : TON_10ms; (*Timeout for read response*)
	UsbNodeListGet_0 : UsbNodeListGet; (*Type of FUB UsbNodeListGet*)
	UsbNodeGet_0 : UsbNodeGet; (*Type of FUB UsbNodeGet*)
	FRM_xopen_0 : FRM_xopen;
	FRM_write_0 : FRM_write;
	FRM_read_0 : FRM_read;
	FRM_rbuf_0 : FRM_rbuf;
	FRM_robuf_0 : FRM_robuf;
	FRM_close_0 : FRM_close;
	ArUserSetPassword_0 : ArUserSetPassword;
	ArUserSetToken_0 : ArUserSetToken;
	ArUserAuthToken_0 : ArUserAuthenticateToken;
END_VAR
(*----------------------------------------------------------------------------------------------------------------------------------------------------------------------------------------------------------------------------------------------------------------------*)
(*Local variables*)
VAR
	rfid_state : rfidManagementEnum := IdleRFID; (*State machine for RFID readet*)
	rfid_init : USINT; (*Init state*)
	callback : rfidManagementEnum; (*Return state after write*)
	usb_data : ARRAY[0..4] OF usbNode_typ; (*Data of all available USB devices*)
	usb_data_linked : usbNode_typ; (*Data of the linked device*)
	data_write : STRING[80]; (*Write data buffer*)
	data_read : STRING[80]; (*Read data buffer*)
	node_id_buffer : ARRAY[0..4] OF UDINT; (*Different nodeIDs saved in array-elements*)
	node : USINT; (*Node number*)
	idx : USINT;
	tmpTokenOld : STRING[80];
	ArUserNameLen : UDINT;
	ArUserNameAdr : UDINT;
	ArUserPasswordLen : UDINT;
	ArUserPasswordAdr : UDINT;
END_VAR
(*----------------------------------------------------------------------------------------------------------------------------------------------------------------------------------------------------------------------------------------------------------------------*)
(*RFID configuration and constants*)
VAR
	DEV_PRODUCT_ID : ARRAY[0..1] OF UINT := [24577,17]; (*1=5E9010.29, 2=5E9030.29*)
	DEV_VENDOR_ID : ARRAY[0..1] OF UINT := [1027,8137]; (*1=5E9010.29, 2=5E9030.29*)
	CFG_ACTIVE : ARRAY[0..9] OF STRING[30];
	REQ_ACTIVE : STRING[30];
END_VAR
VAR CONSTANT
	CFG_5E9010_29 : ARRAY[0..3] OF STRING[30] := ['010A0003041800260000','010C00030410002101000000','0109000304F0000000','0109000304F1FF0000']; (*Reset to Ready, set protocol, set AGC, set receiver mode*)
	REQ_5E9010_29 : STRING[30] := '010B000304140401000000'; (*Acquire the unique token ID*)
	CFG_5E9030_29 : ARRAY[0..4] OF STRING[30] := ['Life',3(' '),''];
END_VAR
(*----------------------------------------------------------------------------------------------------------------------------------------------------------------------------------------------------------------------------------------------------------------------*)
(*Error Constants*)
VAR CONSTANT
	ERR_RFID_BUFFER : DINT := 50000; (*Read response exceeds maximum buffer size*)
	ERR_RFID_RESPONSE : DINT := 50010; (*RFID response incorrect*)
	ERR_RFID_READ_TIMEOUT : DINT := 50020; (*Read response timeout*)
	ERR_RFID_DISCONNECTED : DINT := 50030; (*RFID reader was disconnected*)
END_VAR
```

### changelog.txt
```
Version 0.8
- Update user managment to version 0.8
- Added support for RFID reader 5E9030

Version 0.7
- Clear password field when user is created, password is changed, login or logout
- Removed user anonymous from user list
- Increased length of status message

Version 0.6
- Added message box before deleting user
- Changed constant to avoid conflict with other samples
- Fixed user selection after create and rename
- Updated mappView to 5.7.1
- Code optimizations

Version 0.5
- Code cleanup

Version 0.5
- Multi client support
- Changed error structure

Version 0.4
- Software structure change to work with future expansion
- Make sure passwords match before user is created
- Added support for RFID reader

Version 0.3
- Automatically set password when new user is created
- Erase password field when user logs out
- New command to rename user

Version 0.2
- Make sure last user can not be deleted
- Make sure last user can not delete himself
- Make sure last user can not be deleted
- Added group box with login
- Added message boxes for success and failed commands
- Visual tweaks and bugfixes

Version 0.1
- First public release
```

### Program Logical/UserManagement (IEC)

#### Main.st - Init, cyclic, exit code
```iecst
// --------------------------------------------------------------------------------------------------------------------
// General user task. This is a support task for the mappView visualization. The following functions are implemneted
// - Create and delete user
// - Create and delete roles
// - Change password and assign roles to users
// Version 0.1
// --------------------------------------------------------------------------------------------------------------------
PROGRAM _INIT
	ArUser.PAR.FilePath := 'c:\Temp\UserDataExport.txt';			// Where to export user data
	ArUser.PAR.NumberOfUsers := SIZEOF(ArUser.DAT.Users)/SIZEOF(ArUser.DAT.Users[0]);
END_PROGRAM

PROGRAM _CYCLIC

	// --------------------------------------------------------------------------------------------------------------------
	// Main state machine
	// --------------------------------------------------------------------------------------------------------------------
	CASE UserManagementState OF
		// --------------------------------------------------------------------------------------------------------------------
		// Idle state
		// --------------------------------------------------------------------------------------------------------------------
		IdleState:
			// --------------------------------------------------------------------------------------------------------------------
			// Create role list for current user
			idx := 0;
			brsmemset(ADR(ArUser.VIS.ListUserRole), 0, SIZEOF(ArUser.VIS.ListUserRole));
			WHILE brsstrcmp(ADR(ArUser.DAT.Users[ArUser.VIS.ListUserIndex].Roles[idx]), ADR('')) <> 0 DO
				ArUser.VIS.ListUserRole[idx] := '{"value":"';
				brsstrcat(ADR(ArUser.VIS.ListUserRole[idx]), ADR(ArUser.DAT.Users[ArUser.VIS.ListUserIndex].Roles[idx]));
				brsstrcat(ADR(ArUser.VIS.ListUserRole[idx]), ADR('","text":"'));
				brsstrcat(ADR(ArUser.VIS.ListUserRole[idx]), ADR(ArUser.DAT.Users[ArUser.VIS.ListUserIndex].Roles[idx]));
				brsstrcat(ADR(ArUser.VIS.ListUserRole[idx]), ADR('"}'));
				idx := idx + 1;
			END_WHILE;

			// --------------------------------------------------------------------------------------------------------------------
			// Wait for new command
			IF  (ArUser.CMD.UserCreate) THEN
				UserCreate_0(Execute := FALSE);
				UserManagementState := CreateUserState;
			ELSIF (ArUser.CMD.RoleAssign) THEN
				UserAssignRole_0(Execute := FALSE);
				UserManagementState := AssignRoleState;
			ELSIF (ArUser.CMD.UserDelete) THEN
				DeleteUser_0(Execute := FALSE);
				UserManagementState := DeleteUserState;
			ELSIF (ArUser.CMD.Export) THEN
				ExportUser_0(Execute := FALSE);
				UserManagementState := ExportListState;
			ELSIF (ArUser.CMD.Import) THEN
				ImportUser_0(Execute := FALSE);
				UserManagementState := ImportListState;
			ELSIF (ArUser.CMD.PasswordChange) THEN
				SetPassword_0(Execute := FALSE);
				UserManagementState := ComparePasswordState;
			ELSIF (ArUser.CMD.ListRefresh) THEN
				UserManagementState := CreateUserListGetFirstState;
			END_IF;

			// --------------------------------------------------------------------------------------------------------------------
			// Reset fields on new command
			IF ArUser.CMD.UserCreate OR ArUser.CMD.UserDelete OR ArUser.CMD.RoleCreate OR ArUser.CMD.RoleCreate OR ArUser.CMD.RoleDelete OR ArUser.CMD.RoleAssign OR ArUser.CMD.PasswordChange OR ArUser.CMD.ListRefresh OR ArUser.CMD.Import OR ArUser.CMD.Export OR ArUser.CMD.ErrorReset THEN
				ArUser.DAT.Status := '';
			END_IF;

		// --------------------------------------------------------------------------------------------------------------------
		// Create new user
		// --------------------------------------------------------------------------------------------------------------------
		CreateUserState:
			UserCreate_0(Execute := TRUE , UserName := ArUser.PAR.UserName);

			// --------------------------------------------------------------------------------------------------------------------
			// Success
			IF UserCreate_0.Done AND NOT UserCreate_0.Busy THEN
				ArUser.DAT.Status := 'User created';
				ArUser.CMD.UserCreate := FALSE;
				UserManagementState := CreateUserListGetFirstState;
			// Error
			ELSIF UserCreate_0.Error THEN
				ArUser.ERR.Number := UserCreate_0.ErrorID;
				ArUser.ERR.State := UserManagementState;
				UserManagementState := ErrorState;
			END_IF;

		// --------------------------------------------------------------------------------------------------------------------
		// Assign user role
		// --------------------------------------------------------------------------------------------------------------------
		AssignRoleState:
			UserAssignRole_0(Execute := TRUE , UserName := ArUser.PAR.UserName , RoleName := ArUser.PAR.UserRole);

//			// --------------------------------------------------------------------------------------------------------------------
			// Success
			IF UserAssignRole_0.Done AND NOT UserAssignRole_0.Busy THEN
				ArUser.DAT.Status := 'Role assigned';
				ArUser.CMD.RoleAssign := FALSE;
				UserManagementState := CreateUserListGetFirstState;
			// Error
			ELSIF UserAssignRole_0.Error THEN
				ArUser.ERR.Number := UserAssignRole_0.ErrorID;
				ArUser.ERR.State := UserManagementState;
				UserManagementState := ErrorState;
			END_IF;

		// --------------------------------------------------------------------------------------------------------------------
		// Delete user
		// --------------------------------------------------------------------------------------------------------------------
		DeleteUserState:
			DeleteUser_0(Execute := TRUE , UserName := ArUser.PAR.UserName);

			// --------------------------------------------------------------------------------------------------------------------
			// Success
			IF DeleteUser_0.Done AND NOT DeleteUser_0.Busy THEN
				ArUser.DAT.Status := 'User deleted';
				ArUser.CMD.UserDelete := FALSE;
				UserManagementState := CreateUserListGetFirstState;
			// Error
			ELSIF DeleteUser_0.Error THEN
				ArUser.ERR.Number := DeleteUser_0.ErrorID;
				ArUser.ERR.State := UserManagementState;
				UserManagementState := ErrorState;
			END_IF;

		// --------------------------------------------------------------------------------------------------------------------
		// Export user list to file
		// --------------------------------------------------------------------------------------------------------------------
		ExportListState:
			ExportUser_0(Execute := TRUE , FilePath := ArUser.PAR.FilePath);

			// --------------------------------------------------------------------------------------------------------------------
			// Success
			IF ExportUser_0.Done AND NOT ExportUser_0.Busy THEN
				ArUser.DAT.Status := 'Export finished';
				ArUser.CMD.Export := FALSE;
				UserManagementState := IdleState;
			ELSIF ExportUser_0.Error THEN
				ArUser.ERR.Number := ExportUser_0.ErrorID;
				ArUser.ERR.State := UserManagementState;
				UserManagementState := ErrorState;
			END_IF;

		// --------------------------------------------------------------------------------------------------------------------
		// Import user list from file
		// --------------------------------------------------------------------------------------------------------------------
		ImportListState:
			ImportUser_0(Execute := TRUE , FilePath := ArUser.PAR.FilePath);

			// --------------------------------------------------------------------------------------------------------------------
			// Success
			IF ImportUser_0.Done AND NOT ImportUser_0.Busy THEN
				ArUser.DAT.Status := 'Import finished';
				ArUser.CMD.Import := FALSE;
				UserManagementState := CreateUserListGetFirstState;
			ELSIF ImportUser_0.Error THEN
				ArUser.ERR.Number := ImportUser_0.ErrorID;
				ArUser.ERR.State := UserManagementState;
				UserManagementState := ErrorState;
			END_IF;

		// --------------------------------------------------------------------------------------------------------------------
		// Change password, make sure both passwords are correct
		// --------------------------------------------------------------------------------------------------------------------
		ComparePasswordState:
			IF brsstrcmp(ADR(ArUser.PAR.Password), ADR(ArUser.PAR.PasswordRepeat)) = 0 THEN
				UserManagementState := ChangePasswordState;
			ELSE
				ArUser.ERR.Number := ERR_PASSWORD_MISMATCH;
				ArUser.ERR.State := UserManagementState;
				UserManagementState := ErrorState;
			END_IF;

		// --------------------------------------------------------------------------------------------------------------------
		// Change password, execute password change
		// --------------------------------------------------------------------------------------------------------------------
		ChangePasswordState:
			SetPassword_0(Execute := TRUE , UserName := ArUser.PAR.UserName , Password := ArUser.PAR.Password );

			// --------------------------------------------------------------------------------------------------------------------
			// Success
			IF SetPassword_0.Done AND NOT SetPassword_0.Busy THEN
				ArUser.DAT.Status := 'Password changed!';
				ArUser.CMD.PasswordChange := FALSE;
				UserManagementState := IdleState;
			ELSIF SetPassword_0.Error THEN
				ArUser.ERR.Number := SetPassword_0.ErrorID;
				ArUser.ERR.State := UserManagementState;
				UserManagementState := ErrorState;
			END_IF;

		// --------------------------------------------------------------------------------------------------------------------
		// Create list of users and roles
		// --------------------------------------------------------------------------------------------------------------------
		CreateUserListGetFirstState:
			// Initialize user list
			ArUserInitList_0(Execute := TRUE, ListType := USER_LISTTYPE, ElementName :='');

			// --------------------------------------------------------------------------------------------------------------------
			// Get first user name
			IF ArUserInitList_0.Done AND NOT ArUserInitList_0.Busy THEN
				ArUserGetFirst_0(Execute := TRUE , List := ArUserInitList_0.List );

				// --------------------------------------------------------------------------------------------------------------------
				// Success
				IF ArUserGetFirst_0.Done THEN
					// Clear data, store user name and generate data provider for vis
					brsmemset(ADR(ArUser.DAT.Users), 0, SIZEOF(ArUser.DAT.Users));
					brsmemset(ADR(ArUser.VIS.ListUsers), 0, SIZEOF(ArUser.VIS.ListUsers));
					brsmemset(ADR(ArUser.VIS.ListRoles), 0, SIZEOF(ArUser.VIS.ListRoles));
					UserCounter := 0;

					ArUser.DAT.Users[UserCounter].Name := ArUserGetFirst_0.ElementName;
					ArUser.VIS.ListUsers[UserCounter] := '{"value":"';
					brsstrcat(ADR(ArUser.VIS.ListUsers[UserCounter]), ADR(ArUserGetFirst_0.ElementName));
					brsstrcat(ADR(ArUser.VIS.ListUsers[UserCounter]), ADR('","text":"'));
					brsstrcat(ADR(ArUser.VIS.ListUsers[UserCounter]), ADR(ArUserGetFirst_0.ElementName));
					brsstrcat(ADR(ArUser.VIS.ListUsers[UserCounter]), ADR('"}'));

					// Reset function block and init counters
					ArUserGetFirst_0(Execute := FALSE);
					UserCounter := 1;
					RoleCounter := 0;
					UserManagementState := CreateUserListGetNextState;
					// Error
				ELSIF ArUserGetFirst_0.Error THEN
					ArUser.ERR.Number := ArUserGetFirst_0.ErrorID;
					ArUser.ERR.State := UserManagementState;
					UserManagementState := ErrorState;
				END_IF;
			END_IF;

		CreateUserListGetNextState:
			// Make sure we have space left
			IF UserCounter < ArUser.PAR.NumberOfUsers THEN
				// Get next user
				ArUserGetNext_0(Execute := TRUE , List := ArUserInitList_0.List);

				// --------------------------------------------------------------------------------------------------------------------
				// Success
				IF ArUserGetNext_0.Done THEN
					// Store user name and generate data provider for vis
					ArUser.DAT.Users[UserCounter].Name := ArUserGetNext_0.ElementName;
					ArUser.VIS.ListUsers[UserCounter] := '{"value":"';
					brsstrcat(ADR(ArUser.VIS.ListUsers[UserCounter]), ADR(ArUserGetNext_0.ElementName));
					brsstrcat(ADR(ArUser.VIS.ListUsers[UserCounter]), ADR('","text":"'));
					brsstrcat(ADR(ArUser.VIS.ListUsers[UserCounter]), ADR(ArUserGetNext_0.ElementName));
					brsstrcat(ADR(ArUser.VIS.ListUsers[UserCounter]), ADR('"}'));
					// Reset function block and get next name
					ArUserGetNext_0(Execute := FALSE , List := ArUserInitList_0.List);
					UserCounter := UserCounter + 1;
				// Error
				ELSIF ArUserGetNext_0.Error AND NOT (ArUserGetNext_0.ErrorID = END_OF_LIST) THEN
					ArUser.ERR.Number := ArUserGetNext_0.ErrorID;
					ArUser.ERR.State := UserManagementState;
					UserManagementState := ErrorState;
				// List is complete
				ELSIF ArUserGetNext_0.ErrorID = END_OF_LIST THEN
					// Reset function blocks and counters
					ArUserGetNext_0(Execute := FALSE);
					ArUserGetFirst_0(Execute := FALSE);
					ArUserInitList_0(Execute := FALSE);
					UserCounter := 0;
					RoleCounter := 0;
					UserManagementState := RoleListInitListState;
				END_IF;
//			ELSE
//				ArUser.ERR.Number := ArUserGetNext_0.ErrorID;
//				ArUser.ERR.State := UserManagementState;
//				UserManagementState := ErrorState;
			END_IF;

		// --------------------------------------------------------------------------------------------------------------------
		// Create table of roles assigned to the table of users
		// --------------------------------------------------------------------------------------------------------------------
		RoleListInitListState:
			IF UserCounter < ArUser.PAR.NumberOfUsers XOR (ArUserGetNext_0.ErrorID = END_OF_LIST) THEN
				ArUserInitList_0(Execute := TRUE, ListType := USERROLE_LISTTYPE , ElementName := ArUser.DAT.Users[UserCounter].Name);

				// --------------------------------------------------------------------------------------------------------------------
				// Success
				IF ArUserInitList_0.Done  AND NOT ArUserInitList_0.Busy THEN
					ArUserGetFirst_0(Execute := TRUE , List := ArUserInitList_0.List);
					ArUser.DAT.Users[UserCounter].Roles[0] := ArUserGetFirst_0.ElementName;
					ArUserGetFirst_0(Execute := FALSE , List := ArUserInitList_0.List);
					RoleCounter := 1;
					UserManagementState:= RoleListGetNextState;
				// Error
				ELSIF ArUserInitList_0.Error THEN
					IF ArUserInitList_0.ErrorID = ELEMENT_DOES_NOT_EXIST THEN
						ArUserInitList_0(Execute := FALSE, ListType :=USERROLE_LISTTYPE , ElementName :=ArUser.DAT.Users[UserCounter].Name );
						ArUserGetFirst_0(Execute := FALSE , List := ArUserInitList_0.List);
						UserCounter := 1;
						RoleCounter := 0;
						UserManagementState := CreateRoleListGetFirstState;
					ELSE
						ArUser.ERR.Number := ArUserInitList_0.ErrorID;
						ArUser.ERR.State := UserManagementState;
						UserManagementState := ErrorState;
					END_IF;
				END_IF;
			ELSE

//				UserManagementState := CreateRoleListGetFirstState;
			END_IF;

		RoleListGetNextState:
			ArUserGetNext_0(Execute := TRUE, List := ArUserInitList_0.List);

			// --------------------------------------------------------------------------------------------------------------------
			// Success
			IF ArUserGetNext_0.Done THEN
				ArUser.DAT.Users[UserCounter].Roles[RoleCounter] := ArUserGetNext_0.ElementName;
				ArUserGetNext_0(Execute := FALSE, List := ArUserInitList_0.List);
//				UserCounter := UserCounter + 1;
				RoleCounter := RoleCounter + 1;
			// List is complete
			ELSIF ArUserGetNext_0.ErrorID = END_OF_LIST THEN
				UserCounter := UserCounter + 1;
				ArUserGetNext_0(Execute := FALSE, List := ArUserInitList_0.List);
				ArUserInitList_0(Execute := FALSE, ListType :=USERROLE_LISTTYPE , ElementName :=ArUser.DAT.Users[UserCounter].Name );
				UserManagementState := RoleListInitListState;
			// Error
			ELSIF ArUserGetNext_0.Error THEN
				ArUser.ERR.Number := ArUserGetNext_0.ErrorID;
				ArUser.ERR.State := UserManagementState;
				UserManagementState := ErrorState;
			END_IF;

		// --------------------------------------------------------------------------------------------------------------------
		// Create table of roles
		// --------------------------------------------------------------------------------------------------------------------
		CreateRoleListGetFirstState:
			ArUserInitList_0(Execute := TRUE, ListType := ROLE_LISTTYPE , ElementName :='' );

			// --------------------------------------------------------------------------------------------------------------------
			// Success
			IF ArUserInitList_0.Done AND NOT ArUserInitList_0.Busy THEN
				ArUserGetFirst_0(Execute := TRUE , List := ArUserInitList_0.List );

				// --------------------------------------------------------------------------------------------------------------------
				// Success
				IF ArUserGetFirst_0.Done THEN
					// Store role names and generate data provider for vis
					ArUser.DAT.Roles[RoleCounter] := ArUserGetFirst_0.ElementName;
					ArUser.VIS.ListRoles[RoleCounter] := '{"value":"';
					brsstrcat(ADR(ArUser.VIS.ListRoles[RoleCounter]), ADR(ArUserGetFirst_0.ElementName));
					brsstrcat(ADR(ArUser.VIS.ListRoles[RoleCounter]), ADR('","text":"'));
					brsstrcat(ADR(ArUser.VIS.ListRoles[RoleCounter]), ADR(ArUserGetFirst_0.ElementName));
					brsstrcat(ADR(ArUser.VIS.ListRoles[RoleCounter]), ADR('"}'));
					// Reset function block and init counters
					ArUserGetFirst_0(Execute := FALSE);
					RoleCounter := 1;
					UserManagementState := CreateRoleListGetNextState;
				// Error
				ELSIF ArUserGetFirst_0.Error THEN
					ArUser.ERR.Number := ArUserGetFirst_0.ErrorID;
					ArUser.ERR.State := UserManagementState;
					UserManagementState := ErrorState;
				END_IF;
			// Error
			ELSIF ArUserInitList_0.Error THEN
				ArUser.ERR.Number := ArUserInitList_0.ErrorID;
				ArUser.ERR.State := UserManagementState;
				UserManagementState := ErrorState;
			END_IF;

		CreateRoleListGetNextState:
			IF UserCounter < ArUser.PAR.NumberOfUsers THEN
				ArUserGetNext_0(Execute := TRUE , List := ArUserInitList_0.List);

				// --------------------------------------------------------------------------------------------------------------------
				// Success
				IF ArUserGetNext_0.Done THEN
					// Store user name and generate data provider for vis
					ArUser.DAT.Roles[RoleCounter] := ArUserGetNext_0.ElementName;
					ArUser.VIS.ListRoles[RoleCounter] := '{"value":"';
					brsstrcat(ADR(ArUser.VIS.ListRoles[RoleCounter]), ADR(ArUserGetNext_0.ElementName));
					brsstrcat(ADR(ArUser.VIS.ListRoles[RoleCounter]), ADR('","text":"'));
					brsstrcat(ADR(ArUser.VIS.ListRoles[RoleCounter]), ADR(ArUserGetNext_0.ElementName));
					brsstrcat(ADR(ArUser.VIS.ListRoles[RoleCounter]), ADR('"}'));
					// Reset function block and get next name
					ArUserGetNext_0(Execute := FALSE);
					RoleCounter := RoleCounter + 1;
				// Error
				ELSIF ArUserGetNext_0.Error AND NOT (ArUserGetNext_0.ErrorID = END_OF_LIST) THEN
					ArUser.ERR.Number := ArUserGetNext_0.ErrorID;
					ArUser.ERR.State := UserManagementState;
					UserManagementState := ErrorState;
				// End of list reached
				ELSIF ArUserGetNext_0.ErrorID = END_OF_LIST THEN
					ArUserGetNext_0(Execute := FALSE);
					ArUserGetFirst_0(Execute := FALSE);
					ArUserInitList_0(Execute := FALSE);
					RoleCounter := 0;
					ArUser.CMD.ListRefresh := FALSE;
					UserManagementState := IdleState;
				END_IF;
			ELSE
//				UserManagementState := IdleState;
			END_IF;

		// --------------------------------------------------------------------------------------------------------------------
		// Error state
		// --------------------------------------------------------------------------------------------------------------------
		ErrorState:
			// --------------------------------------------------------------------------------------------------------------------
			// Generate text for most common errors
			IF(ArUser.ERR.Number = arUSER_ERR_ALREADY_EXISTS) THEN
				ArUser.DAT.Status := 'ERR: User/Role already exists';
			ELSIF(ArUser.ERR.Number = arUSER_ERR_PARAMETER) THEN
				ArUser.DAT.Status := 'ERR: User/Role is empty';
			ELSIF(ArUser.ERR.Number = arUSER_ERR_DOES_NOT_EXIST) THEN
				ArUser.DAT.Status := 'ERR: User/Role does not exist';
			ELSIF(ArUser.ERR.Number = ERR_PASSWORD_MISMATCH) THEN
				ArUser.DAT.Status := 'ERR: Passwords do not match';
			END_IF
			// --------------------------------------------------------------------------------------------------------------------
			// Return to idle state
			IF ArUser.CMD.ErrorReset THEN
				ArUser.DAT.Status := '';

				UserCounter := 1;
				RoleCounter := 0;

				brsmemset(ADR(ArUser.ERR), 0, SIZEOF(ArUser.ERR));
				ArUser.CMD.ErrorReset := FALSE;
				UserManagementState := IdleState;
			END_IF;
			brsmemset(ADR(ArUser.CMD), 0, SIZEOF(ArUser.CMD));
	END_CASE;
END_PROGRAM
```

#### Types.typ - Local data types
```iecst
TYPE
	typUSER : 	STRUCT
		CMD : typUSER_CMD;
		PAR : typUSER_PAR;
		DAT : typUSER_DAT;
		VIS : typUSER_VIS;
		ERR : typUSER_ERR;
	END_STRUCT;
	typUSER_CMD : 	STRUCT
		UserCreate : BOOL;
		UserDelete : BOOL;
		PasswordChange : BOOL;
		RoleCreate : BOOL;
		RoleDelete : BOOL;
		RoleAssign : BOOL;
		Import : BOOL;
		Export : BOOL;
		ListRefresh : BOOL;
		ErrorReset : BOOL;
	END_STRUCT;
	typUSER_PAR : 	STRUCT
		FilePath : STRING[80];
		UserName : STRING[80];
		UserRole : STRING[80];
		Password : STRING[80];
		PasswordRepeat : STRING[80];
		NumberOfUsers : USINT;
		AssignRole : STRING[128];
		AssignRoleName : STRING[128];
	END_STRUCT;
	typUSER_DAT : 	STRUCT
		Users : ARRAY[0..49]OF typUSER_DETAILS;
		Roles : ARRAY[0..19]OF STRING[80];
		Status : STRING[80];
	END_STRUCT;
	typUSER_VIS : 	STRUCT
		New_Member : USINT;
	END_STRUCT;
	typUSER_ERR : 	STRUCT
		Number : DINT;
		State : UserManagementEnum;
	END_STRUCT;
	typUSER_DETAILS : 	STRUCT
		Roles : ARRAY[0..9]OF STRING[80];
		Name : STRING[80];
	END_STRUCT;
	UserManagementEnum :
		(
		IdleState,
		DestroyListState,
		CreateUserState,
		DeleteUserState,
		ExportListState,
		ImportListState,
		ChangePasswordState,
		ComparePasswordState,
		CreateUserListGetNextState,
		CreateUserListGetFirstState,
		AssignRoleState,
		RoleListMainState,
		RoleListDeleteListState,
		RoleListInitListState,
		ErrorState,
		CreateRoleListGetFirstState,
		CreateRoleListGetNextState,
		RoleListGetNextState
		);
END_TYPE
```

#### Variables.var - Local variables
```iecst
(*General*)
VAR
	UserManagementState : UserManagementEnum := IdleState; (*State Machine for UserManagementState*)
	UserCreate_0 : ArUserCreate; (*UserCreate -> Create an user with given name; default no password *)
	DeleteUser_0 : ArUserDelete; (*UserDelete -> Delete an user  *)
	ExportUser_0 : ArUserExport;
	ImportUser_0 : ArUserImport;
	SetPassword_0 : ArUserSetPassword;
	UserAssignRole_0 : ArUserAssignRole;
	ArUserGetNext_0 : ArUserGetNext;
	ArUserGetFirst_0 : ArUserGetFirst;
	ArUserInitList_0 : ArUserInitList;
	ArUserDestroyList_0 : ArUserDestroyList;
	tmpStr : STRING[80];
	idx : USINT;
END_VAR
(*Loop counter*)
VAR
	RoleCounter : USINT; (*LoopCounter for creating the table; 1 = second element of array*)
	UserCounter : USINT;
END_VAR
(*List types *)
VAR CONSTANT
	USER_LISTTYPE : BYTE := 1; (*List Type User*)
	ROLE_LISTTYPE : BYTE := 2; (*List Type Role*)
	USERROLE_LISTTYPE : BYTE := 3; (*List Type UserRole*)
END_VAR
(*Error Constants*)
VAR CONSTANT
	ERR_PASSWORD_MISMATCH : DINT := 50000;
	END_OF_LIST : DINT := -2144327714;
	ELEMENT_DOES_NOT_EXIST : DINT := -1070585892;
END_VAR
```

#### changelog.txt
```
Version 0.3
- Automatically set password when new user is created
- Erase password field when user logs out
- New command to rename user

Version 0.2
- Make sure last user can not be deleted
- Make sure last user can not delete himself
- Make sure last user can not be deleted
- Added group box with login
- Added message boxes for success and failed commands
- Visual tweaks and bugfixes

Version 0.1
- First public release
```

Listed in the project but not available here: Logical/mappUser/UserManagement/Types.typ, Logical/mappUser/UserManagement/LocalFunctions.st
